# EPICS substitutions: HVCAENx527App/Db/HVCAENx527.substitutions
file "$(TOP)/templates/HVCAENx527.tpl" {
	pattern {PSNAME}
	{ "\$(P):\$(PSNAME)" }
}
